FUNCTION_BLOCK FB_Add
VAR_INPUT	
	iIn1,iIn2: INT;
END_VAR
VAR_OUTPUT
	iOut: INT;
END_VAR
VAR
END_VAR

 iOut := iIn1+iIn2;

END_FUNCTION_BLOCK

(* stored: Version 1.1.0.1, ProductVersion 3.1.4024.12
   POU FB_Add: Id {8087d907-4094-4b49-bdd5-b69edb00538e}, SpecialFunc None *)
